// TIA Portal V20 export
DATA_BLOCK "BK34"   // DB309
// stored: MemoryReserve 100
   VAR
      "X10-1.UNWINDER #1 RADIUS MEASURE" : Bool := FALSE;
      "X10-2.UNWINDER #2 RADIUS MEASURE" : Bool := FALSE;
      "X12-1.SPARE" : Bool := FALSE;
      "X12-2.SPARE" : Bool := FALSE;
      "X14-1.SPARE" : Bool := FALSE;
      "X14-2.SPARE" : Bool := FALSE;
      "X16-1.SPARE" : Bool := FALSE;
      "X16-2.SPARE" : Bool := FALSE;
   END_VAR
BEGIN
END_DATA_BLOCK
